TYPE ST_GroupElement_HMI :
STRUCT
	bZmiennaGroupElement	: BOOL;
	
END_STRUCT
END_TYPE

(* stored: Version 1.1.0.1, ProductVersion 3.1.4024.15
   DUT ST_GroupElement_HMI: Id {9a71b668-6ecf-4c4c-912c-2910233f1c9c} *)
